SUBAPPLICATION Zaehler (* Subapplication Type *)
  (* Standard: 61499-2 *)
  (* Version 1.0, 2023-02-17, Franz *)
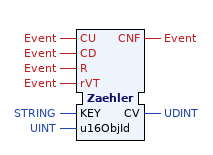
  EVENT_INPUT
    CU; (* Count Up *)
    CD; (* Count Down *)
    R; (* Reset *)
    rVT; (* refresh VT *)
  END_EVENT
  EVENT_OUTPUT
    CNF; (* Confirmation -- Counter Value was changed *)
  END_EVENT
  VAR_INPUT
    KEY : STRING;
    u16ObjId : UINT;
  END_VAR
  VAR_OUTPUT
    CV : UDINT; (* Counter Value *)
  END_VAR
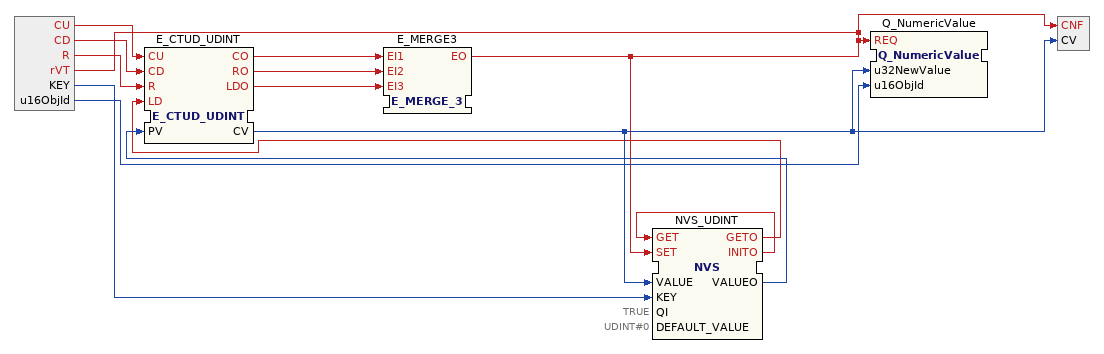
  FBS
    E_CTUD_UDINT : E_CTUD_UDINT;
    Q_NumericValue : Q_NumericValue;
    NVS_UDINT : NVS(QI := TRUE, DEFAULT_VALUE := UDINT#0);
    E_MERGE3 : E_MERGE_3;
  END_FBS
  EVENT_CONNECTIONS
    CU TO E_CTUD_UDINT.CU;
    CD TO E_CTUD_UDINT.CD;
    R TO E_CTUD_UDINT.R;
    rVT TO Q_NumericValue.REQ;
    rVT TO CNF;
    NVS_UDINT.GETO TO E_CTUD_UDINT.LD;
    NVS_UDINT.INITO TO NVS_UDINT.GET;
    E_CTUD_UDINT.CO TO E_MERGE3.EI1;
    E_CTUD_UDINT.RO TO E_MERGE3.EI2;
    E_CTUD_UDINT.LDO TO E_MERGE3.EI3;
    E_MERGE3.EO TO NVS_UDINT.SET;
    E_MERGE3.EO TO CNF;
    E_MERGE3.EO TO Q_NumericValue.REQ;
  END_CONNECTIONS
  DATA_CONNECTIONS
    E_CTUD_UDINT.CV TO Q_NumericValue.u32NewValue;
    E_CTUD_UDINT.CV TO CV;
    u16ObjId TO Q_NumericValue.u16ObjId;
    E_CTUD_UDINT.CV TO NVS_UDINT.VALUE;
    NVS_UDINT.VALUEO TO E_CTUD_UDINT.PV;
    KEY TO NVS_UDINT.KEY;
  END_CONNECTIONS
END_SUBAPPLICATION
